FUNCTION_BLOCK FB_RetainTimer
VAR_INPUT
	Enable 		: BOOL;			// Enable timer
	Reset 		: BOOL;			// Reset timer
END_VAR
VAR_OUTPUT
	ET			: TIME := T#0S;	// Elapsed TIME
	ET_ms		: DWORD;		// Elapsed DWORD milliseconds
END_VAR
VAR
	RTRIG_Enable	: R_TRIG;
	FTRIG_Enable	: F_TRIG;
	RTRIG_Reset		: R_TRIG;
	StartTime		: TIME := T#0S;
	SessionTime		: TIME := T#0S;
	TotalTime		: TIME := T#0S;
END_VAR

RTRIG_Enable(CLK := Enable);
FTRIG_Enable(CLK := Enable);
RTRIG_Reset(CLK := Reset);

// RESET
	IF(RTRIG_Reset.Q) THEN
		StartTime 	:= T#0S;
		SessionTime := T#0S;
		TotalTime 	:= T#0S;
	END_IF

// ENABLE
	IF(RTRIG_Enable.Q AND NOT Reset) THEN
		StartTime := TIME();
	END_IF
	
	IF(FTRIG_Enable.Q) THEN
		TotalTime := TotalTime + SessionTime;
		SessionTime := T#0s;
	END_IF

///////////////////////////////////////////////////////////////

// Updating time
IF(Enable AND NOT Reset) THEN
	SessionTime := TIME() - StartTime;
END_IF

ET := TotalTime + SessionTime;
ET_ms := TIME_TO_DWORD(ET);

END_FUNCTION_BLOCK

(* stored: Version 1.1.0.1, ProductVersion 3.1.4024.13
   POU FB_RetainTimer: Id {5f9d101b-b15e-442c-8c53-76ff9dc9e749}, SpecialFunc None *)
